// TIA Portal V18 export
// export: Created 2026-06-12T00:00:00Z, ExportSetting WithDefaults
VAR_GLOBAL   // PLC tag table "AI_PLC_Tags_CIP_Mixing"
   AI_LT3203_PV AT %MD200 : Real;   // Mức bồn trộn 1 LT3203 (0.0 đến 1000.0 L)
   AI_TT3204_PV AT %MD204 : Real;   // Nhiệt độ bồn trộn 1 TT3204 (0.0 đến 100.0 °C)
   AI_LT3209_PV AT %MD208 : Real;   // Mức bồn trộn 2 LT3209 (0.0 đến 1000.0 L)
   AI_TT3208_PV AT %MD212 : Real;   // Nhiệt độ bồn trộn 2 TT3208 (0.0 đến 100.0 °C)
   AI_LT3213_PV AT %MD216 : Real;   // Mức bồn trộn 3 LT3213 (0.0 đến 1000.0 L)
   AI_TT3214_PV AT %MD220 : Real;   // Nhiệt độ bồn trộn 3 TT3214 (0.0 đến 100.0 °C)
   AI_LT3218_PV AT %MD224 : Real;   // Mức bồn trộn 4 LT3218 (0.0 đến 1000.0 L)
   AI_TT3219_PV AT %MD228 : Real;   // Nhiệt độ bồn trộn 4 TT3219 (0.0 đến 100.0 °C)
   AI_BON1_Chay AT %M232.0 : Bool;   // Báo trạng thái bồn trộn 1 đang chạy
   AI_BON2_Chay AT %M232.1 : Bool;   // Báo trạng thái bồn trộn 2 đang chạy
   AI_BON3_Chay AT %M232.2 : Bool;   // Báo trạng thái bồn trộn 3 đang chạy
   AI_BON4_Chay AT %M232.3 : Bool;   // Báo trạng thái bồn trộn 4 đang chạy
   AI_PUMP3264_Chay AT %M232.4 : Bool;   // Trạng thái chạy của bơm PUMP3264
   AI_PUMP3265_Chay AT %M232.5 : Bool;   // Trạng thái chạy của bơm PUMP3265
   AI_Logged_In AT %MW234 : Int;   // Trạng thái đăng nhập trên HMI
   Sim_Counter AT %MD236 : Real;   // Biến đếm trung gian cho sóng tam giác mô phỏng
   Sim_Dir AT %M240.0 : Bool;   // Bit hướng đếm mô phỏng (0: Tăng, 1: Giảm)
   Sim_Val_Norm AT %MD242 : Real;   // Giá trị đếm đã chuẩn hóa về dải 0.0 - 1.0
   Timer_Sim_Pulse_Output AT %M240.1 : Bool;   // Xung kích hoạt đếm từ Timer
END_VAR
